// TIA Portal project "Cau2" (V16)

(* hardware
DEVICE "S7-1200 station_1"  S7-1200 Station
   slot 0: "Rack_0"  S7-1200 Rack  Rack  V1.0
   slot 1: "PLC_1"  CPU 1214C AC/DC/Rly  6ES7 214-1BG40-0XB0  V4.2
*)

// ===== PLC "PLC_1"  CPU 1214C AC/DC/Rly =====

VAR_GLOBAL   // PLC tag table "Default tag table"
   "Tag_1" AT %I1.1 : Bool;
   "Tag_2" AT %I1.0 : Bool;
   "Tag_3" AT %M0.0 : Bool;
   "Tag_4" AT %M0.1 : Bool;
   "Tag_5" AT %M0.4 : Bool;
   "Tag_6" AT %M0.2 : Bool;
   "Tag_7" AT %M0.5 : Bool;
   "M0" AT %Q0.0 : Bool;
   "M3" AT %Q0.1 : Bool;
   "M4" AT %Q0.2 : Bool;
END_VAR

// folder: System blocks/Program resources

DATA_BLOCK "T1"   // DB1
{ S7_Optimized_Access := 'TRUE' }
AUTHOR : Simatic
FAMILY : IEC
NAME : IEC_TMR
VERSION : 1.0
// stored: InstanceOfName IEC_TIMER
"IEC_TIMER"
BEGIN
END_DATA_BLOCK

DATA_BLOCK "T2"   // DB2
{ S7_Optimized_Access := 'TRUE' }
AUTHOR : Simatic
FAMILY : IEC
NAME : IEC_TMR
VERSION : 1.0
// stored: InstanceOfName IEC_TIMER
"IEC_TIMER"
BEGIN
END_DATA_BLOCK

// folder: (top level)

ORGANIZATION_BLOCK "Main"   // OB1, LAD, ProgramCycle
TITLE = "Main Program Sweep (Cycle)"
{ S7_Optimized_Access := 'TRUE' }
VERSION : 0.1
   VAR_INPUT
      Initial_Call : Bool;   // Initial call of this OB
      Remanence : Bool;   // =True, if remanent data are available
   END_VAR
   VAR_TEMP   // added for the SCL form of the ladder/FBD networks
      _w1 : Bool;
   END_VAR
BEGIN

REGION Network 1
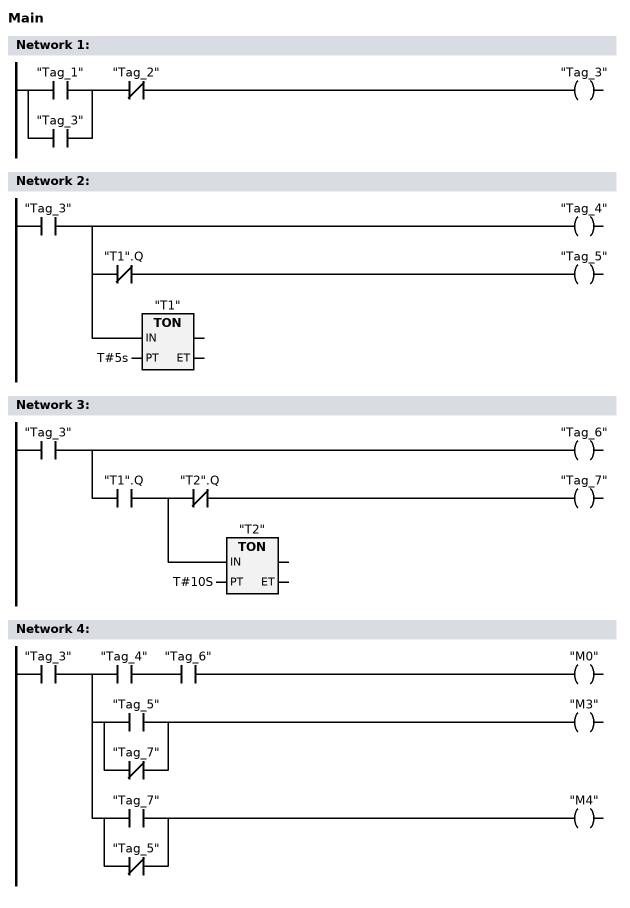
   RUNG wire#powerrail
      Contact( "Tag_1" )
      wire#w1
      I_Contact( "Tag_2" )
      Coil( "Tag_3" )
   END_RUNG
   RUNG wire#powerrail
      Contact( "Tag_3" )
   END_RUNG wire#w1
   // the same network as SCL:
   "Tag_3" := ("Tag_1" OR "Tag_3") AND NOT "Tag_2";
END_REGION

REGION Network 2
   "Tag_4" := "Tag_3";
   "Tag_5" := "Tag_3" AND NOT "T1".Q;
   "T1".TON(IN := "Tag_3", PT := T#5s);
END_REGION

REGION Network 3
   "Tag_6" := "Tag_3";
   #_w1 := "Tag_3" AND "T1".Q;
   "Tag_7" := #_w1 AND NOT "T2".Q;
   "T2".TON(IN := #_w1, PT := T#10S);
END_REGION

REGION Network 4
   RUNG wire#powerrail
      Contact( "Tag_3" )
      wire#w1
      Contact( "Tag_4" )
      Contact( "Tag_6" )
      Coil( "M0" )
   END_RUNG
   RUNG wire#w1
      Contact( "Tag_5" )
      wire#w2
      Coil( "M3" )
   END_RUNG
   RUNG wire#w1
      I_Contact( "Tag_7" )
   END_RUNG wire#w2
   RUNG wire#w1
      Contact( "Tag_7" )
      wire#w3
      Coil( "M4" )
   END_RUNG
   RUNG wire#w1
      I_Contact( "Tag_5" )
   END_RUNG wire#w3
   // the same network as SCL:
   "M0" := "Tag_3" AND "Tag_4" AND "Tag_6";
   "M3" := "Tag_3" AND ("Tag_5" OR NOT "Tag_7");
   "M4" := "Tag_3" AND ("Tag_7" OR NOT "Tag_5");
END_REGION
END_ORGANIZATION_BLOCK